// TIA Portal V17 export
// export: Created 2022-07-16T16:56:09.9496574Z, ExportSetting WithDefaults, DisplayName Totally Integrated Automation Portal, DisplayVersion V17, DisplayName TIA Portal Openness, DisplayVersion V17, DisplayName TIA Portal Version Control Interface, DisplayVersion V17, DisplayName TIA Portal Test Suite Advanced, DisplayVersion V17, DisplayName STEP 7 Professional, DisplayVersion V17, DisplayName STEP 7 Safety, DisplayVersion V17, DisplayName WinCC Professional, DisplayVersion V17
TYPE "connectionParameterType"
// stored: IsFailsafeCompliant false
   STRUCT
      ConnectInfo { ExternalAccessible := 'False'; ExternalVisible := 'False'; ExternalWritable := 'False'; S7_SetPoint := 'True'} : OPC_UA_SessionConnectInfo;
      ConnectionHdl { ExternalAccessible := 'False'; ExternalVisible := 'False'; ExternalWritable := 'False'} : DWord;
      ServerEndpointUrl { ExternalAccessible := 'False'; ExternalVisible := 'False'; ExternalWritable := 'False'} : String[254] := 'opc.tcp://192.168.0.2:4840';
   END_STRUCT;
   // ConnectInfo.SessionName := WSTRING#'OPC UA Connection_1';
   // ConnectInfo.ApplicationName := WSTRING#'';
   // ConnectInfo.SecurityMsgMode := 1;
   // ConnectInfo.SecurityPolicy := 1;
   // ConnectInfo.ServerUri := '';
   // ConnectInfo.CheckServerCertificate := False;
   // ConnectInfo.TransportProfile := 1;
   // ConnectInfo.UserIdentityTokenType := 0;
   // ConnectInfo.CertificateID := 0;
   // ConnectInfo.SessionTimeout := T#30S;
   // ConnectInfo.MonitorConnection := T#5S;
   // ConnectInfo.LocaleIDs[0] := 'en-US';
   // ConnectInfo.LocaleIDs[1..4] := '';
END_TYPE
